(* CoDeSys 2.3 export: _ERR.EXP *)

(* Data type *)
TYPE _ERR :
STRUCT
	State:	       BOOL;
	StateM:		 BOOL;
	Msg:		 STRING[100];
	Zoomer: 	 BOOL;
	Latch:	       BOOL;
	LatchState:   BOOL;
	Lock:           BOOL;
END_STRUCT
END_TYPE
